(*
A circular buffer for storing states.  
*)
FUNCTION_BLOCK INTERNAL _StateBuffer
VAR_GENERIC CONSTANT
	STATE_CAP			: UDINT(1..16#7FFFFFFF) := 1;
END_VAR
VAR
	_iState				: ARRAY[1..STATE_CAP] OF I_StateInternal;
	_nHead				: UDINT := 1;
	_nTail				: UDINT := 1;
	_nLen				: UDINT;
END_VAR

(*
Returns the maximum capacity of the state buffer, indicating how many states it can hold.
*)
METHOD Cap : UDINT
VAR_INPUT
END_VAR
Cap := STATE_CAP;
END_METHOD

(*
Returns the current number of states stored in the buffer.
*)
METHOD Length : UDINT
VAR_INPUT
END_VAR
Length := _nLen;
END_METHOD

(*
Removes and retrieves the oldest state from the buffer.  

Returns:
- `Ok` - If a state is successfully removed.
- `None` - If the buffer is empty.
*)
METHOD Pop : Result
VAR_OUTPUT
	iState			: I_StateInternal;
END_VAR
IF _nHead = _nTail THEN
    Pop := None;
    RETURN;
END_IF

iState := _iState[_nHead];
_iState[_nHead] := 0;

_nHead := _nHead + 1;
_nLen := _nLen - 1;

IF _nHead > STATE_CAP THEN
    _nHead := 1;
END_IF

Pop := Ok;
END_METHOD

(*
Adds a new state to the buffer.  
Returns:
- `Ok` - If the state is successfully added.
- `Err.Itf0` - If the provided state interface is invalid.
- `Err.Ovf` - If the buffer is full.
*)
METHOD Push : Result
VAR_INPUT
	iState			: I_StateInternal;
END_VAR
VAR
	_nNextTail 		: UDINT;
END_VAR
IF iState = 0 THEN
	Push := Err.Itf0;
	RETURN;
END_IF

_nNextTail := _nTail + 1;

IF _nNextTail > STATE_CAP THEN
    _nNextTail := 1;
END_IF

IF _nNextTail = _nHead THEN
    Push := Err.Ovf; 
    RETURN;
END_IF

_nLen := _nLen + 1;
_iState[_nTail] := iState;
_nTail := _nNextTail;
Push := Ok;
END_METHOD

END_FUNCTION_BLOCK

(* stored: Version 1.1.0.1
   POU _StateBuffer: Id {711a25fc-792a-4435-9ccd-e8054980130d}, SpecialFunc None
   Folder Other: Id {5d3df489-8735-43fe-a81c-03404c1c5f20}
   Folder Push: Id {4903ac7f-b709-435c-851d-d394b1e3ffec}
   Method Cap: Id {0d43e644-fff4-43e2-a039-01aede7b9e10}
   Method Length: Id {264889a2-4c66-4869-80d2-31916bbd4e00}
   Method Pop: Id {d39e1d8e-6957-40eb-ad12-24d995eb484b}
   Method Push: Id {5955ea9d-3baf-4dfd-a5a1-a995221ac391} *)
